// TIA Portal V17 export
// export: Created 2025-06-26T07:11:12.1198651Z, ExportSetting WithDefaults, DisplayName Totally Integrated Automation Portal, DisplayVersion V17 Update 8, DisplayName TIA Portal Openness, DisplayVersion V17 Update 8, DisplayName TIA Portal Version Control Interface, DisplayVersion V17, DisplayName STEP 7 Professional, DisplayVersion V17 Update 8, DisplayName STEP 7 Safety, DisplayVersion V17 Update 6, DisplayName WinCC Advanced, DisplayVersion V17 Update 8
VAR_GLOBAL   // PLC tag table "Auxiliary_IO"
   Rack2Slot20_I AT %I310.0 : "stET200AL_AQ_I";   //    {ExternalAccessible false, ExternalVisible false, ExternalWritable false}
   Rack2Slot21_I AT %I320.0 : "stET200AL_AI";   //    {ExternalAccessible false, ExternalVisible false, ExternalWritable false}
   Rack1Slot9_I AT %I170.0 : "stET200AL_AI";   //    {ExternalAccessible false, ExternalVisible false, ExternalWritable false}
   Rack1Slot8_I AT %I160.0 : "stET200AL_AI";   //    {ExternalAccessible false, ExternalVisible false, ExternalWritable false}
   Rack1Slot7_I AT %I150.0 : "stET200AL_AI";   //    {ExternalAccessible false, ExternalVisible false, ExternalWritable false}
   Rack2Slot25_I AT %I360.0 : "stET200AL_AI";   //    {ExternalAccessible false, ExternalVisible false, ExternalWritable false}
   Rack1Slot5_I AT %I130.0 : "stET200AL_AI";   //    {ExternalAccessible false, ExternalVisible false, ExternalWritable false}
   Rack1Slot4_I AT %I120.0 : "stET200AL_RTD";   //    {ExternalAccessible false, ExternalVisible false, ExternalWritable false}
   Rack1Slot6_I AT %I140.0 : "stET200AL_AI";   //    {ExternalAccessible false, ExternalVisible false, ExternalWritable false}
   Rack2Slot19_I AT %I300.0 : "stET200AL_AI";   //    {ExternalAccessible false, ExternalVisible false, ExternalWritable false}
   Rack1Slot2_I AT %I100.0 : "stET200AL_AI";   //    {ExternalAccessible false, ExternalVisible false, ExternalWritable false}
   Rack2Slot23_I AT %I340.0 : "stET200AL_AI";   //    {ExternalAccessible false, ExternalVisible false, ExternalWritable false}
   Rack2Slot22_I AT %I330.0 : "stET200AL_AI";   //    {ExternalAccessible false, ExternalVisible false, ExternalWritable false}
   Rack1Slot3_I AT %I110.0 : "stET200AL_RTD";   //    {ExternalAccessible false, ExternalVisible false, ExternalWritable false}
   Rack2Slot24_I AT %I350.0 : "stET200AL_AI";   //    {ExternalAccessible false, ExternalVisible false, ExternalWritable false}
   Rack2Slot29_I AT %I400.0 : "stET200AL_AI";   //    {ExternalAccessible false, ExternalVisible false, ExternalWritable false}
   Rack2Slot30_I AT %I410.0 : "stET200AL_AI";   //    {ExternalAccessible false, ExternalVisible false, ExternalWritable false}
   Rack2Slot31_I AT %I420.0 : "stET200AL_AI";   //    {ExternalAccessible false, ExternalVisible false, ExternalWritable false}
   Rack2Slot32_I AT %I430.0 : "stET200AL_RTD";   //    {ExternalAccessible false, ExternalVisible false, ExternalWritable false}
   Rack2Slot33_I AT %I440.0 : "stET200AL_AI";   //    {ExternalAccessible false, ExternalVisible false, ExternalWritable false}
   Rack2Slot34_I AT %I450.0 : "stET200AL_AI";   //    {ExternalAccessible false, ExternalVisible false, ExternalWritable false}
   Rack2Slot26_I AT %I370.0 : "stET200AL_AQ_I";   //    {ExternalAccessible false, ExternalVisible false, ExternalWritable false}
   Rack2Slot27_I AT %I380.0 : "stET200AL_AI";   //    {ExternalAccessible false, ExternalVisible false, ExternalWritable false}
   Rack2Slot28_I AT %I390.0 : "stET200AL_AQ_I";   //    {ExternalAccessible false, ExternalVisible false, ExternalWritable false}
   Rack2Slot20_Q AT %Q310.0 : "stET200AL_AQ";   //    {ExternalAccessible false, ExternalVisible false, ExternalWritable false}
   Rack2Slot21_Q AT %Q320.0 : "stET200AL_AQ";   //    {ExternalAccessible false, ExternalVisible false, ExternalWritable false}
   Rack1Slot10_I AT %I180.0 : "stET200AL_DIQ_I";   //    {ExternalAccessible false, ExternalVisible false, ExternalWritable false}
   Rack1Slot11_I AT %I190.0 : "stET200AL_RTD";   //    {ExternalAccessible false, ExternalVisible false, ExternalWritable false}
   Rack1Slot12_I AT %I200.0 : "stET200AL_AI";   //    {ExternalAccessible false, ExternalVisible false, ExternalWritable false}
   Rack1Slot13_I AT %I210.0 : "stET200AL_AI";   //    {ExternalAccessible false, ExternalVisible false, ExternalWritable false}
   Rack1Slot14_I AT %I248.0 : "stET200AL_RTD";   //    {ExternalAccessible false, ExternalVisible false, ExternalWritable false}
   Rack1Slot15_I AT %I230.0 : "stET200AL_AI";   //    {ExternalAccessible false, ExternalVisible false, ExternalWritable false}
   Rack1Slot16_I AT %I240.0 : "stET200AL_AI";   //    {ExternalAccessible false, ExternalVisible false, ExternalWritable false}
   Rack1Slot17_I AT %I250.0 : "stET200AL_AI";   //    {ExternalAccessible false, ExternalVisible false, ExternalWritable false}
   Rack2Slot19_Q AT %Q300.0 : "stET200AL_AQ";   //    {ExternalAccessible false, ExternalVisible false, ExternalWritable false}
   Rack2Slot22_Q AT %Q330.0 : "stET200AL_AQ";   //    {ExternalAccessible false, ExternalVisible false, ExternalWritable false}
   Rack2Slot23_Q AT %Q340.0 : "stET200AL_AQ";   //    {ExternalAccessible false, ExternalVisible false, ExternalWritable false}
   Rack2Slot24_Q AT %Q350.0 : "stET200AL_AQ";   //    {ExternalAccessible false, ExternalVisible false, ExternalWritable false}
   Rack2Slot25_Q AT %Q360.0 : "stET200AL_AQ";   //    {ExternalAccessible false, ExternalVisible false, ExternalWritable false}
   Rack2Slot26_Q AT %Q370.0 : "stET200AL_AQ";   //    {ExternalAccessible false, ExternalVisible false, ExternalWritable false}
   Rack2Slot27_Q AT %Q380.0 : "stET200AL_AQ";   //    {ExternalAccessible false, ExternalVisible false, ExternalWritable false}
   Rack2Slot28_Q AT %Q390.0 : "stET200AL_AQ";   //    {ExternalAccessible false, ExternalVisible false, ExternalWritable false}
   Rack2Slot29_Q AT %Q400.0 : "stET200AL_AQ";   //    {ExternalAccessible false, ExternalVisible false, ExternalWritable false}
   Rack2Slot30_Q AT %Q410.0 : "stET200AL_AQ";   //    {ExternalAccessible false, ExternalVisible false, ExternalWritable false}
   Rack2Slot31_Q AT %Q420.0 : "stET200AL_AQ";   //    {ExternalAccessible false, ExternalVisible false, ExternalWritable false}
   Rack2Slot32_Q AT %Q430.0 : "stET200AL_AQ";   //    {ExternalAccessible false, ExternalVisible false, ExternalWritable false}
   Rack2Slot33_Q AT %Q440.0 : "stET200AL_AQ";   //    {ExternalAccessible false, ExternalVisible false, ExternalWritable false}
   Rack2Slot34_Q AT %Q450.0 : "stET200AL_AQ";   //    {ExternalAccessible false, ExternalVisible false, ExternalWritable false}
   Rack1Slot10_Q AT %Q180.0 : "stET200AL_DIQ_Q";   //    {ExternalAccessible false, ExternalVisible false, ExternalWritable false}
END_VAR
